// TIA Portal V20 export
TYPE "UDT_AnaAccu"
TITLE = MTPDataObjectSUCLibrary/DataAssembly/AccuView
   STRUCT
      WQC { ExternalWritable := 'False'} : Byte := 16#FF;   // Worst Quality Code variable
      AcCnt1 { ExternalWritable := 'False'} : Real := 0.0;   // Accumulated counter #1
      AcCnt2 { ExternalWritable := 'False'} : Real := 0.0;   // Accumulated counter #2
      AcCntUnit { ExternalWritable := 'False'} : Int := 1001;   // Unit of AcCnt1 / AcCnt2
   END_STRUCT;
END_TYPE
